// Mitsubishi GX Works2 project: 42015005-기말1   PLC: Q02/Q02H

PROGRAM MAIN
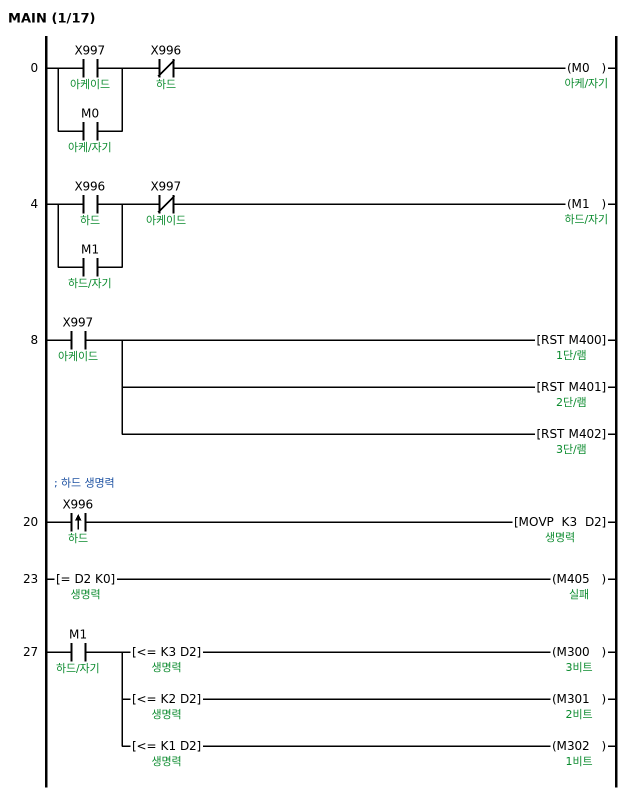
0     LD      X997  ; 아케이드
      OR      M0  ; 아케/자기
      ANI     X996  ; 하드
      OUT     M0  ; 아케/자기
4     LD      X996  ; 하드
      OR      M1  ; 하드/자기
      ANI     X997  ; 아케이드
      OUT     M1  ; 하드/자기
8     LD      X997  ; 아케이드
      RST     M400  ; 1단/램
      RST     M401  ; 2단/램
      RST     M402  ; 3단/램
; 하드 생명력
20    LDP     X996  ; 하드
      MOVP    K3 D2  ; 생명력
23    LD=     D2 K0  ; 생명력
      OUT     M405  ; 실패
27    LD      M1  ; 하드/자기
      MPS
      AND<=   K3 D2  ; 생명력
      OUT     M300  ; 3비트
      MRD
      AND<=   K2 D2  ; 생명력
      OUT     M301  ; 2비트
      MPP
      AND<=   K1 D2  ; 생명력
      OUT     M302  ; 1비트
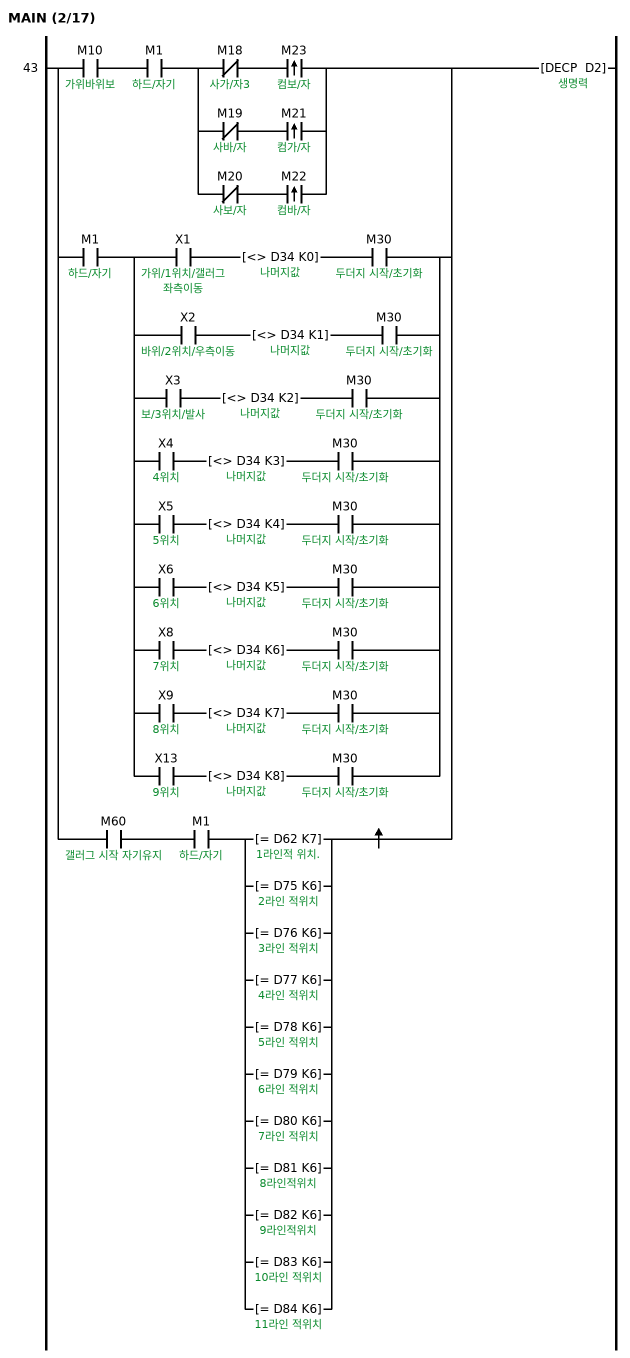
43    LD      M10  ; 가위바위보
      AND     M1  ; 하드/자기
      LDI     M18  ; 사가/자3
      ANDP    M23  ; 컴보/자
      LDI     M19  ; 사바/자
      ANDP    M21  ; 컴가/자
      ORB
      LDI     M20  ; 사보/자
      ANDP    M22  ; 컴바/자
      ORB
      ANB
      LD      M1  ; 하드/자기
      LD      X1  ; 가위/1위치/갤러그 좌측이동
      AND<>   D34 K0  ; 나머지값
      AND     M30  ; 두더지 시작/초기화
      LD      X2  ; 바위/2위치/우측이동
      AND<>   D34 K1  ; 나머지값
      AND     M30  ; 두더지 시작/초기화
      ORB
      LD      X3  ; 보/3위치/발사
      AND<>   D34 K2  ; 나머지값
      AND     M30  ; 두더지 시작/초기화
      ORB
      LD      X4  ; 4위치
      AND<>   D34 K3  ; 나머지값
      AND     M30  ; 두더지 시작/초기화
      ORB
      LD      X5  ; 5위치
      AND<>   D34 K4  ; 나머지값
      AND     M30  ; 두더지 시작/초기화
      ORB
      LD      X6  ; 6위치
      AND<>   D34 K5  ; 나머지값
      AND     M30  ; 두더지 시작/초기화
      ORB
      LD      X8  ; 7위치
      AND<>   D34 K6  ; 나머지값
      AND     M30  ; 두더지 시작/초기화
      ORB
      LD      X9  ; 8위치
      AND<>   D34 K7  ; 나머지값
      AND     M30  ; 두더지 시작/초기화
      ORB
      LD      X13  ; 9위치
      AND<>   D34 K8  ; 나머지값
      AND     M30  ; 두더지 시작/초기화
      ORB
      ANB
      ORB
      LD      M60  ; 갤러그 시작 자기유지
      AND     M1  ; 하드/자기
      LD=     D62 K7  ; 1라인적 위치.
      OR=     D75 K6  ; 2라인 적위치
      OR=     D76 K6  ; 3라인 적위치
      OR=     D77 K6  ; 4라인 적위치
      OR=     D78 K6  ; 5라인 적위치
      OR=     D79 K6  ; 6라인 적위치
      OR=     D80 K6  ; 7라인 적위치
      OR=     D81 K6  ; 8라인적위치
      OR=     D82 K6  ; 9라인적위치
      OR=     D83 K6  ; 10라인 적위치
      OR=     D84 K6  ; 11라인 적위치
      ANB
      MEP
      ORB
      DECP    D2
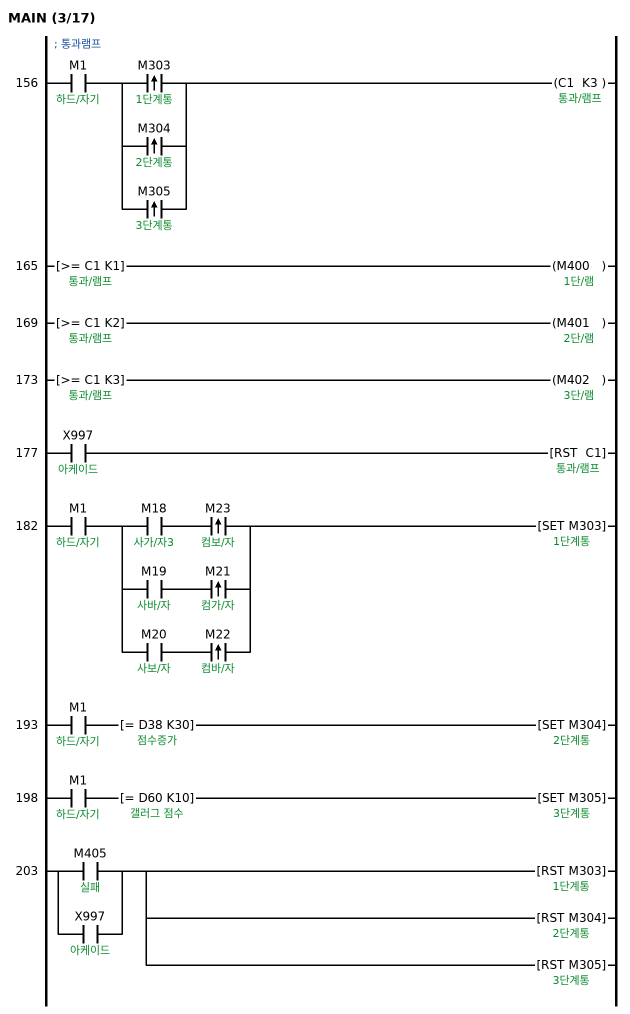
; 통과램프
156   LD      M1  ; 하드/자기
      LDP     M303  ; 1단계통
      ORP     M304  ; 2단계통
      ORP     M305  ; 3단계통
      ANB
      OUT     C1 K3  ; 통과/램프
165   LD>=    C1 K1  ; 통과/램프
      OUT     M400  ; 1단/램
169   LD>=    C1 K2  ; 통과/램프
      OUT     M401  ; 2단/램
173   LD>=    C1 K3  ; 통과/램프
      OUT     M402  ; 3단/램
177   LD      X997  ; 아케이드
      RST     C1  ; 통과/램프
182   LD      M1  ; 하드/자기
      LD      M18  ; 사가/자3
      ANDP    M23  ; 컴보/자
      LD      M19  ; 사바/자
      ANDP    M21  ; 컴가/자
      ORB
      LD      M20  ; 사보/자
      ANDP    M22  ; 컴바/자
      ORB
      ANB
      SET     M303  ; 1단계통
193   LD      M1  ; 하드/자기
      AND=    D38 K30  ; 점수증가
      SET     M304  ; 2단계통
198   LD      M1  ; 하드/자기
      AND=    D60 K10  ; 갤러그 점수
      SET     M305  ; 3단계통
203   LD      M405  ; 실패
      OR      X997  ; 아케이드
      RST     M303  ; 1단계통
      RST     M304  ; 2단계통
      RST     M305  ; 3단계통
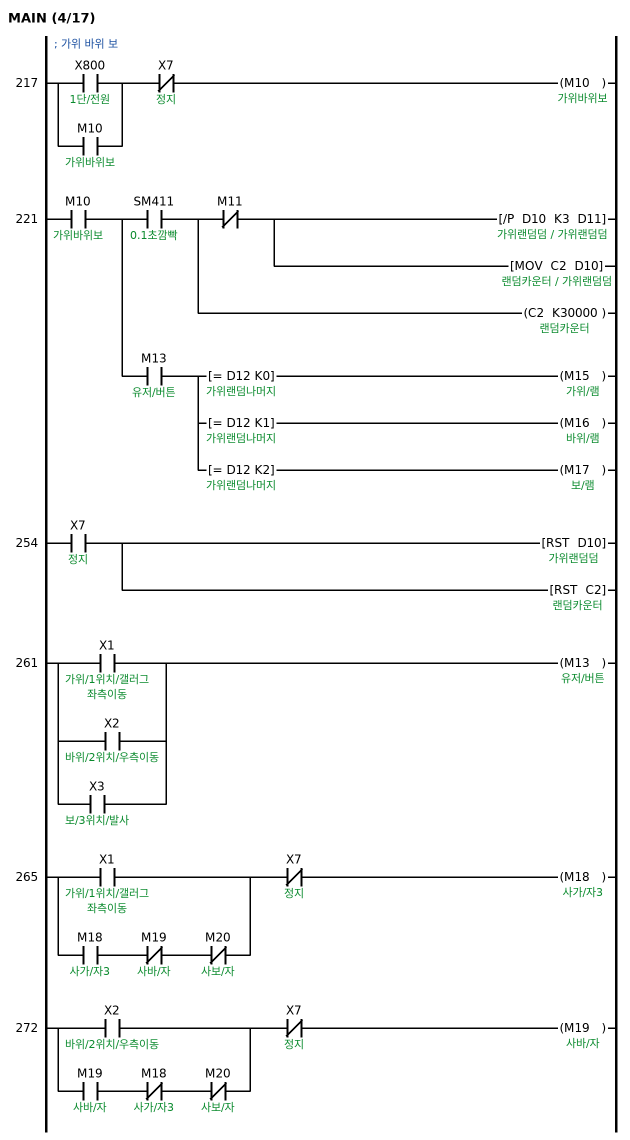
; 가위 바위 보
217   LD      X800  ; 1단/전원
      OR      M10  ; 가위바위보
      ANI     X7  ; 정지
      OUT     M10  ; 가위바위보
221   LD      M10  ; 가위바위보
      MPS
      AND     SM411  ; 0.1초깜빡
      MPS
      ANI     M11
      /P      D10 K3 D11  ; 가위랜덤덤 / 가위랜덤덤
      MOV     C2 D10  ; 랜덤카운터
      MPP
      OUT     C2 K30000  ; 랜덤카운터
      MPP
      AND     M13  ; 유저/버튼
      MPS
      AND=    D12 K0  ; 가위랜덤나머지
      OUT     M15  ; 가위/램
      MRD
      AND=    D12 K1  ; 가위랜덤나머지
      OUT     M16  ; 바위/램
      MPP
      AND=    D12 K2  ; 가위랜덤나머지
      OUT     M17  ; 보/램
254   LD      X7  ; 정지
      RST     D10  ; 가위랜덤덤
      RST     C2  ; 랜덤카운터
261   LD      X1  ; 가위/1위치/갤러그 좌측이동
      OR      X2  ; 바위/2위치/우측이동
      OR      X3  ; 보/3위치/발사
      OUT     M13  ; 유저/버튼
265   LD      X1  ; 가위/1위치/갤러그 좌측이동
      LD      M18  ; 사가/자3
      ANI     M19  ; 사바/자
      ANI     M20  ; 사보/자
      ORB
      ANI     X7  ; 정지
      OUT     M18  ; 사가/자3
272   LD      X2  ; 바위/2위치/우측이동
      LD      M19  ; 사바/자
      ANI     M18  ; 사가/자3
      ANI     M20  ; 사보/자
      ORB
      ANI     X7  ; 정지
      OUT     M19  ; 사바/자
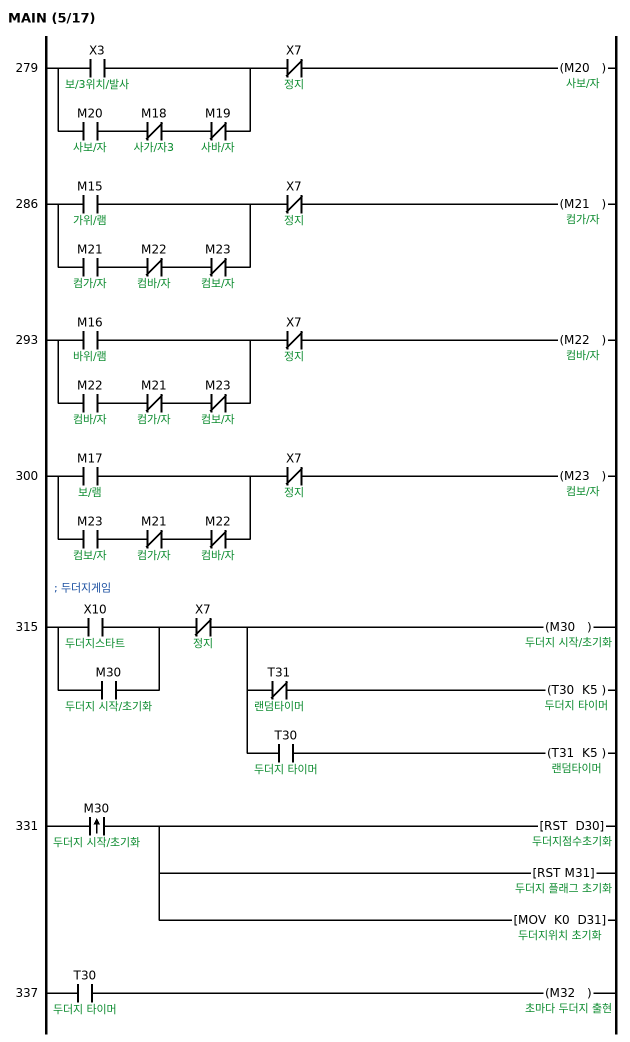
279   LD      X3  ; 보/3위치/발사
      LD      M20  ; 사보/자
      ANI     M18  ; 사가/자3
      ANI     M19  ; 사바/자
      ORB
      ANI     X7  ; 정지
      OUT     M20  ; 사보/자
286   LD      M15  ; 가위/램
      LD      M21  ; 컴가/자
      ANI     M22  ; 컴바/자
      ANI     M23  ; 컴보/자
      ORB
      ANI     X7  ; 정지
      OUT     M21  ; 컴가/자
293   LD      M16  ; 바위/램
      LD      M22  ; 컴바/자
      ANI     M21  ; 컴가/자
      ANI     M23  ; 컴보/자
      ORB
      ANI     X7  ; 정지
      OUT     M22  ; 컴바/자
300   LD      M17  ; 보/램
      LD      M23  ; 컴보/자
      ANI     M21  ; 컴가/자
      ANI     M22  ; 컴바/자
      ORB
      ANI     X7  ; 정지
      OUT     M23  ; 컴보/자
; 두더지게임
315   LD      X10  ; 두더지스타트
      OR      M30  ; 두더지 시작/초기화
      ANI     X7  ; 정지
      OUT     M30  ; 두더지 시작/초기화
      MPS
      ANI     T31  ; 랜덤타이머
      OUT     T30 K5  ; 두더지 타이머
      MPP
      AND     T30  ; 두더지 타이머
      OUT     T31 K5  ; 랜덤타이머
331   LDP     M30  ; 두더지 시작/초기화
      RST     D30  ; 두더지점수초기화
      RST     M31  ; 두더지 플래그 초기화
      MOV     K0 D31  ; 두더지위치 초기화
337   LD      T30  ; 두더지 타이머
      OUT     M32  ; 초마다 두더지 출현
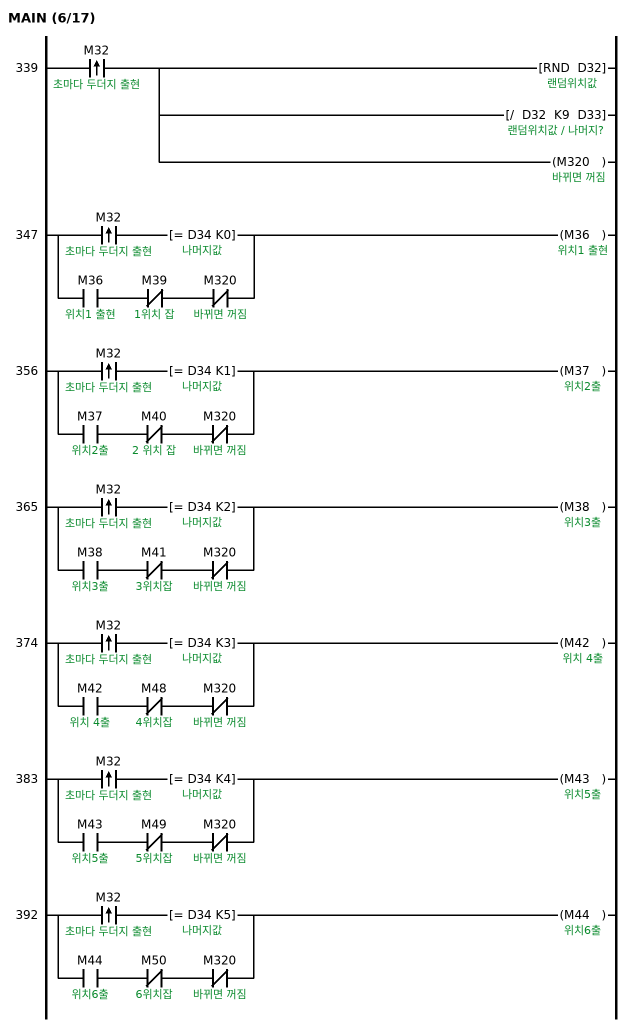
339   LDP     M32  ; 초마다 두더지 출현
      RND     D32  ; 랜덤위치값
      /       D32 K9 D33  ; 나머지?
      OUT     M320  ; 바뀌면 꺼짐
347   LDP     M32  ; 초마다 두더지 출현
      AND=    D34 K0  ; 나머지값
      LD      M36  ; 위치1 출현
      ANI     M39  ; 1위치 잡
      ANI     M320  ; 바뀌면 꺼짐
      ORB
      OUT     M36  ; 위치1 출현
356   LDP     M32  ; 초마다 두더지 출현
      AND=    D34 K1  ; 나머지값
      LD      M37  ; 위치2출
      ANI     M40  ; 2 위치 잡
      ANI     M320  ; 바뀌면 꺼짐
      ORB
      OUT     M37  ; 위치2출
365   LDP     M32  ; 초마다 두더지 출현
      AND=    D34 K2  ; 나머지값
      LD      M38  ; 위치3출
      ANI     M41  ; 3위치잡
      ANI     M320  ; 바뀌면 꺼짐
      ORB
      OUT     M38  ; 위치3출
374   LDP     M32  ; 초마다 두더지 출현
      AND=    D34 K3  ; 나머지값
      LD      M42  ; 위치 4출
      ANI     M48  ; 4위치잡
      ANI     M320  ; 바뀌면 꺼짐
      ORB
      OUT     M42  ; 위치 4출
383   LDP     M32  ; 초마다 두더지 출현
      AND=    D34 K4  ; 나머지값
      LD      M43  ; 위치5출
      ANI     M49  ; 5위치잡
      ANI     M320  ; 바뀌면 꺼짐
      ORB
      OUT     M43  ; 위치5출
392   LDP     M32  ; 초마다 두더지 출현
      AND=    D34 K5  ; 나머지값
      LD      M44  ; 위치6출
      ANI     M50  ; 6위치잡
      ANI     M320  ; 바뀌면 꺼짐
      ORB
      OUT     M44  ; 위치6출
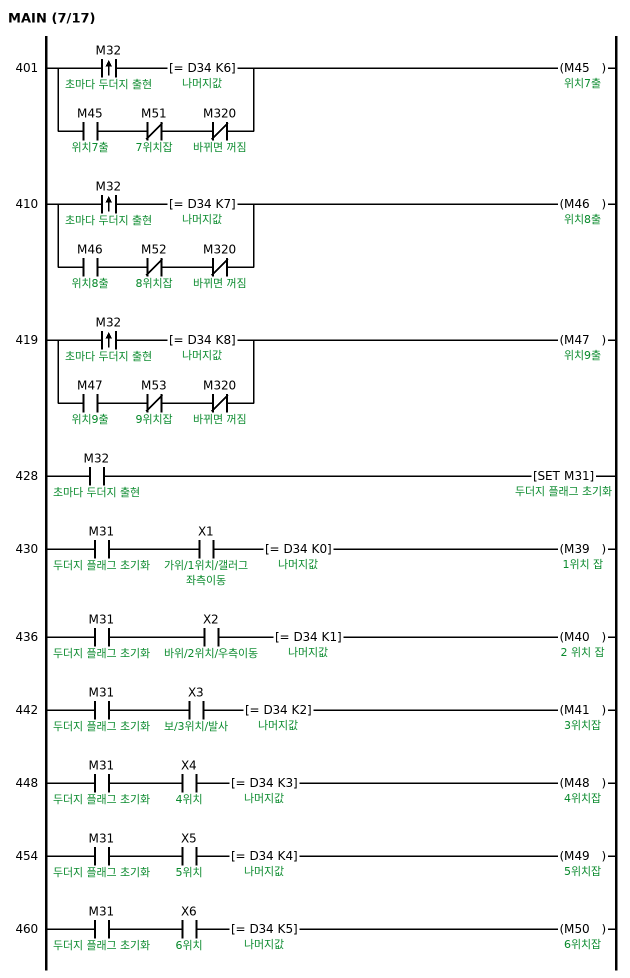
401   LDP     M32  ; 초마다 두더지 출현
      AND=    D34 K6  ; 나머지값
      LD      M45  ; 위치7출
      ANI     M51  ; 7위치잡
      ANI     M320  ; 바뀌면 꺼짐
      ORB
      OUT     M45  ; 위치7출
410   LDP     M32  ; 초마다 두더지 출현
      AND=    D34 K7  ; 나머지값
      LD      M46  ; 위치8출
      ANI     M52  ; 8위치잡
      ANI     M320  ; 바뀌면 꺼짐
      ORB
      OUT     M46  ; 위치8출
419   LDP     M32  ; 초마다 두더지 출현
      AND=    D34 K8  ; 나머지값
      LD      M47  ; 위치9출
      ANI     M53  ; 9위치잡
      ANI     M320  ; 바뀌면 꺼짐
      ORB
      OUT     M47  ; 위치9출
428   LD      M32  ; 초마다 두더지 출현
      SET     M31  ; 두더지 플래그 초기화
430   LD      M31  ; 두더지 플래그 초기화
      AND     X1  ; 가위/1위치/갤러그 좌측이동
      AND=    D34 K0  ; 나머지값
      OUT     M39  ; 1위치 잡
436   LD      M31  ; 두더지 플래그 초기화
      AND     X2  ; 바위/2위치/우측이동
      AND=    D34 K1  ; 나머지값
      OUT     M40  ; 2 위치 잡
442   LD      M31  ; 두더지 플래그 초기화
      AND     X3  ; 보/3위치/발사
      AND=    D34 K2  ; 나머지값
      OUT     M41  ; 3위치잡
448   LD      M31  ; 두더지 플래그 초기화
      AND     X4  ; 4위치
      AND=    D34 K3  ; 나머지값
      OUT     M48  ; 4위치잡
454   LD      M31  ; 두더지 플래그 초기화
      AND     X5  ; 5위치
      AND=    D34 K4  ; 나머지값
      OUT     M49  ; 5위치잡
460   LD      M31  ; 두더지 플래그 초기화
      AND     X6  ; 6위치
      AND=    D34 K5  ; 나머지값
      OUT     M50  ; 6위치잡
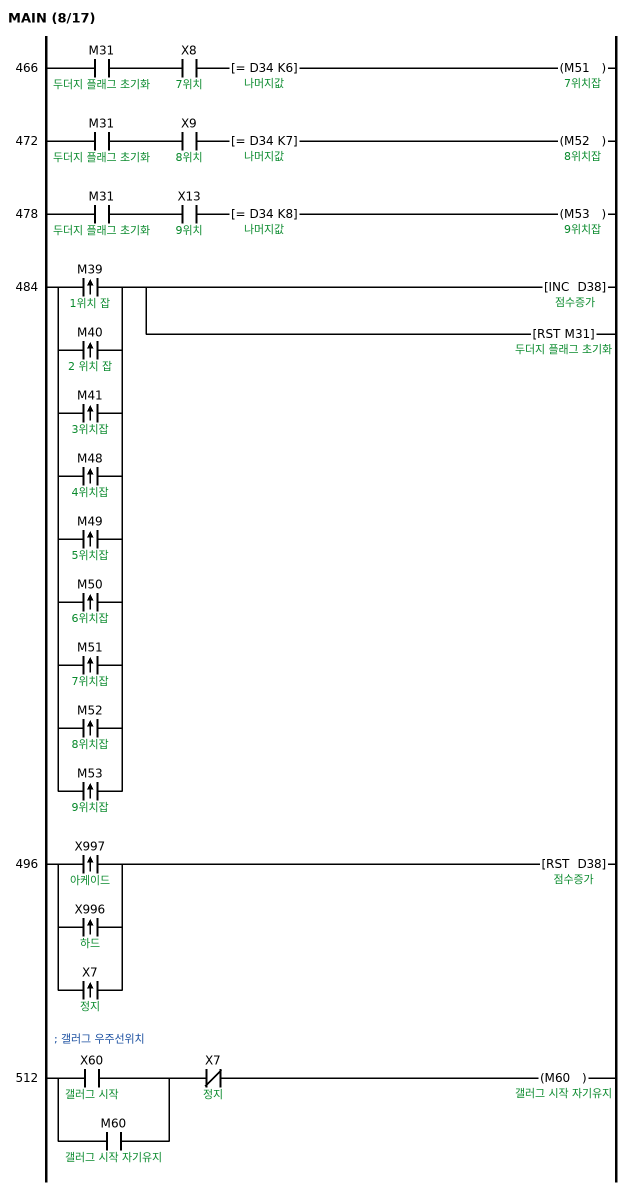
466   LD      M31  ; 두더지 플래그 초기화
      AND     X8  ; 7위치
      AND=    D34 K6  ; 나머지값
      OUT     M51  ; 7위치잡
472   LD      M31  ; 두더지 플래그 초기화
      AND     X9  ; 8위치
      AND=    D34 K7  ; 나머지값
      OUT     M52  ; 8위치잡
478   LD      M31  ; 두더지 플래그 초기화
      AND     X13  ; 9위치
      AND=    D34 K8  ; 나머지값
      OUT     M53  ; 9위치잡
484   LDP     M39  ; 1위치 잡
      ORP     M40  ; 2 위치 잡
      ORP     M41  ; 3위치잡
      ORP     M48  ; 4위치잡
      ORP     M49  ; 5위치잡
      ORP     M50  ; 6위치잡
      ORP     M51  ; 7위치잡
      ORP     M52  ; 8위치잡
      ORP     M53  ; 9위치잡
      INC     D38
      RST     M31  ; 두더지 플래그 초기화
496   LDP     X997  ; 아케이드
      ORP     X996  ; 하드
      ORP     X7  ; 정지
      RST     D38  ; 점수증가
; 갤러그 우주선위치
512   LD      X60  ; 갤러그 시작
      OR      M60  ; 갤러그 시작 자기유지
      ANI     X7  ; 정지
      OUT     M60  ; 갤러그 시작 자기유지
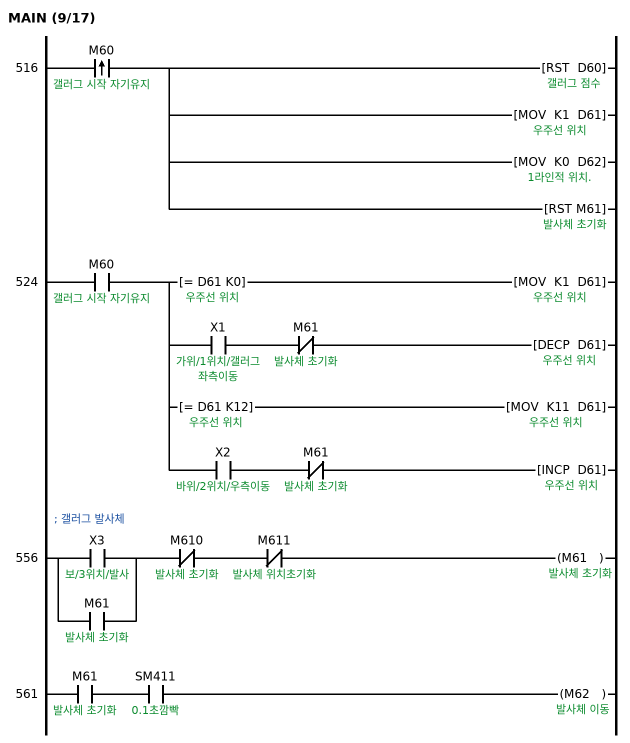
516   LDP     M60  ; 갤러그 시작 자기유지
      RST     D60  ; 갤러그 점수
      MOV     K1 D61  ; 우주선 위치
      MOV     K0 D62
      RST     M61  ; 발사체 초기화
524   LD      M60  ; 갤러그 시작 자기유지
      MPS
      AND=    D61 K0  ; 우주선 위치
      MOV     K1 D61
      MRD
      AND     X1  ; 가위/1위치/갤러그 좌측이동
      ANI     M61  ; 발사체 초기화
      DECP    D61
      MRD
      AND=    D61 K12  ; 우주선 위치
      MOV     K11 D61
      MPP
      AND     X2  ; 바위/2위치/우측이동
      ANI     M61  ; 발사체 초기화
      INCP    D61
; 갤러그 발사체
556   LD      X3  ; 보/3위치/발사
      OR      M61  ; 발사체 초기화
      ANI     M610  ; 발사체 초기화
      ANI     M611  ; 발사체 위치초기화
      OUT     M61  ; 발사체 초기화
561   LD      M61  ; 발사체 초기화
      AND     SM411  ; 0.1초깜빡
      OUT     M62  ; 발사체 이동
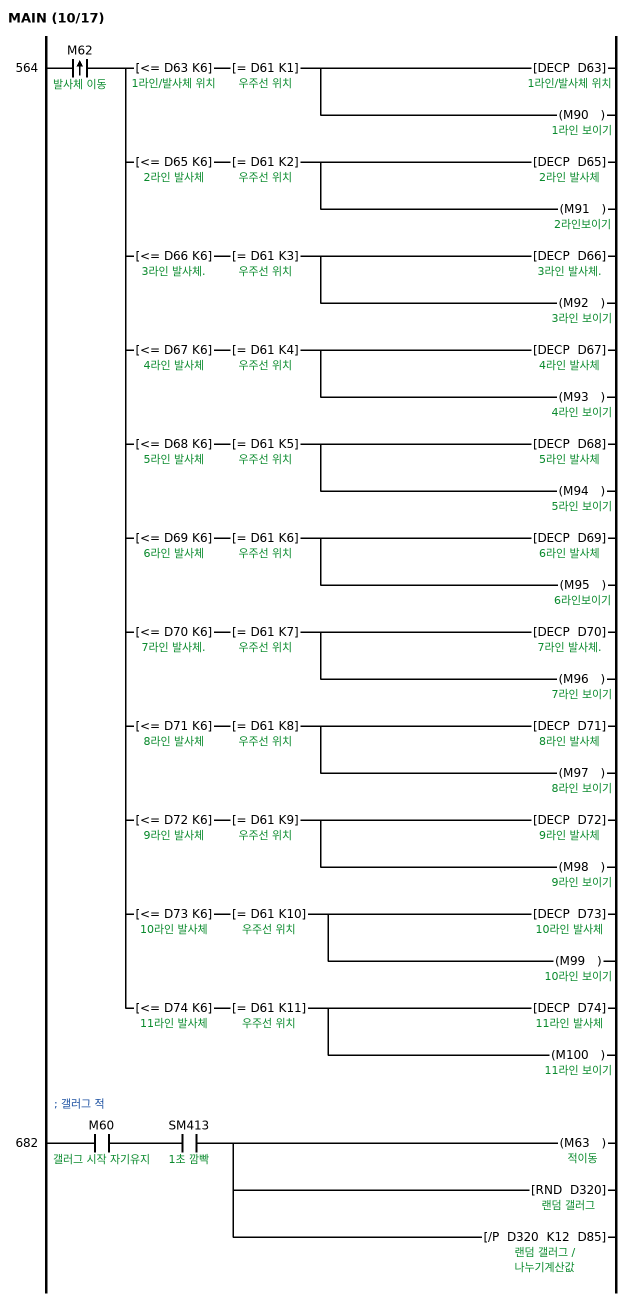
564   LDP     M62  ; 발사체 이동
      MPS
      AND<=   D63 K6  ; 1라인/발사체 위치
      AND=    D61 K1  ; 우주선 위치
      DECP    D63
      OUT     M90  ; 1라인 보이기
      MRD
      AND<=   D65 K6  ; 2라인 발사체
      AND=    D61 K2  ; 우주선 위치
      DECP    D65
      OUT     M91  ; 2라인보이기
      MRD
      AND<=   D66 K6  ; 3라인 발사체.
      AND=    D61 K3  ; 우주선 위치
      DECP    D66
      OUT     M92  ; 3라인 보이기
      MRD
      AND<=   D67 K6  ; 4라인 발사체
      AND=    D61 K4  ; 우주선 위치
      DECP    D67
      OUT     M93  ; 4라인 보이기
      MRD
      AND<=   D68 K6  ; 5라인 발사체
      AND=    D61 K5  ; 우주선 위치
      DECP    D68
      OUT     M94  ; 5라인 보이기
      MRD
      AND<=   D69 K6  ; 6라인 발사체
      AND=    D61 K6  ; 우주선 위치
      DECP    D69
      OUT     M95  ; 6라인보이기
      MRD
      AND<=   D70 K6  ; 7라인 발사체.
      AND=    D61 K7  ; 우주선 위치
      DECP    D70
      OUT     M96  ; 7라인 보이기
      MRD
      AND<=   D71 K6  ; 8라인 발사체
      AND=    D61 K8  ; 우주선 위치
      DECP    D71
      OUT     M97  ; 8라인 보이기
      MRD
      AND<=   D72 K6  ; 9라인 발사체
      AND=    D61 K9  ; 우주선 위치
      DECP    D72
      OUT     M98  ; 9라인 보이기
      MRD
      AND<=   D73 K6  ; 10라인 발사체
      AND=    D61 K10  ; 우주선 위치
      DECP    D73
      OUT     M99  ; 10라인 보이기
      MPP
      AND<=   D74 K6  ; 11라인 발사체
      AND=    D61 K11  ; 우주선 위치
      DECP    D74
      OUT     M100  ; 11라인 보이기
; 갤러그 적
682   LD      M60  ; 갤러그 시작 자기유지
      AND     SM413  ; 1초 깜빡
      OUT     M63  ; 적이동
      RND     D320  ; 랜덤 갤러그
      /P      D320 K12 D85  ; 나누기계산값
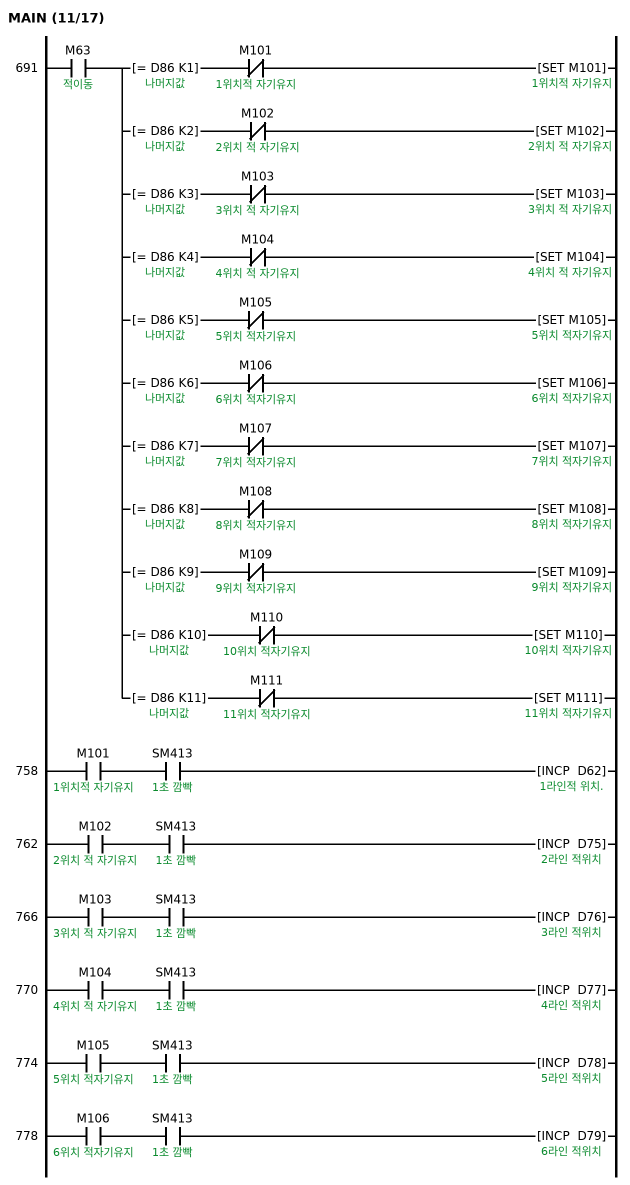
691   LD      M63  ; 적이동
      MPS
      AND=    D86 K1  ; 나머지값
      ANI     M101  ; 1위치적 자기유지
      SET     M101  ; 1위치적 자기유지
      MRD
      AND=    D86 K2  ; 나머지값
      ANI     M102  ; 2위치 적 자기유지
      SET     M102  ; 2위치 적 자기유지
      MRD
      AND=    D86 K3  ; 나머지값
      ANI     M103  ; 3위치 적 자기유지
      SET     M103  ; 3위치 적 자기유지
      MRD
      AND=    D86 K4  ; 나머지값
      ANI     M104  ; 4위치 적 자기유지
      SET     M104  ; 4위치 적 자기유지
      MRD
      AND=    D86 K5  ; 나머지값
      ANI     M105  ; 5위치 적자기유지
      SET     M105  ; 5위치 적자기유지
      MRD
      AND=    D86 K6  ; 나머지값
      ANI     M106  ; 6위치 적자기유지
      SET     M106  ; 6위치 적자기유지
      MRD
      AND=    D86 K7  ; 나머지값
      ANI     M107  ; 7위치 적자기유지
      SET     M107  ; 7위치 적자기유지
      MRD
      AND=    D86 K8  ; 나머지값
      ANI     M108  ; 8위치 적자기유지
      SET     M108  ; 8위치 적자기유지
      MRD
      AND=    D86 K9  ; 나머지값
      ANI     M109  ; 9위치 적자기유지
      SET     M109  ; 9위치 적자기유지
      MRD
      AND=    D86 K10  ; 나머지값
      ANI     M110  ; 10위치 적자기유지
      SET     M110  ; 10위치 적자기유지
      MPP
      AND=    D86 K11  ; 나머지값
      ANI     M111  ; 11위치 적자기유지
      SET     M111  ; 11위치 적자기유지
758   LD      M101  ; 1위치적 자기유지
      AND     SM413  ; 1초 깜빡
      INCP    D62
762   LD      M102  ; 2위치 적 자기유지
      AND     SM413  ; 1초 깜빡
      INCP    D75
766   LD      M103  ; 3위치 적 자기유지
      AND     SM413  ; 1초 깜빡
      INCP    D76
770   LD      M104  ; 4위치 적 자기유지
      AND     SM413  ; 1초 깜빡
      INCP    D77
774   LD      M105  ; 5위치 적자기유지
      AND     SM413  ; 1초 깜빡
      INCP    D78
778   LD      M106  ; 6위치 적자기유지
      AND     SM413  ; 1초 깜빡
      INCP    D79
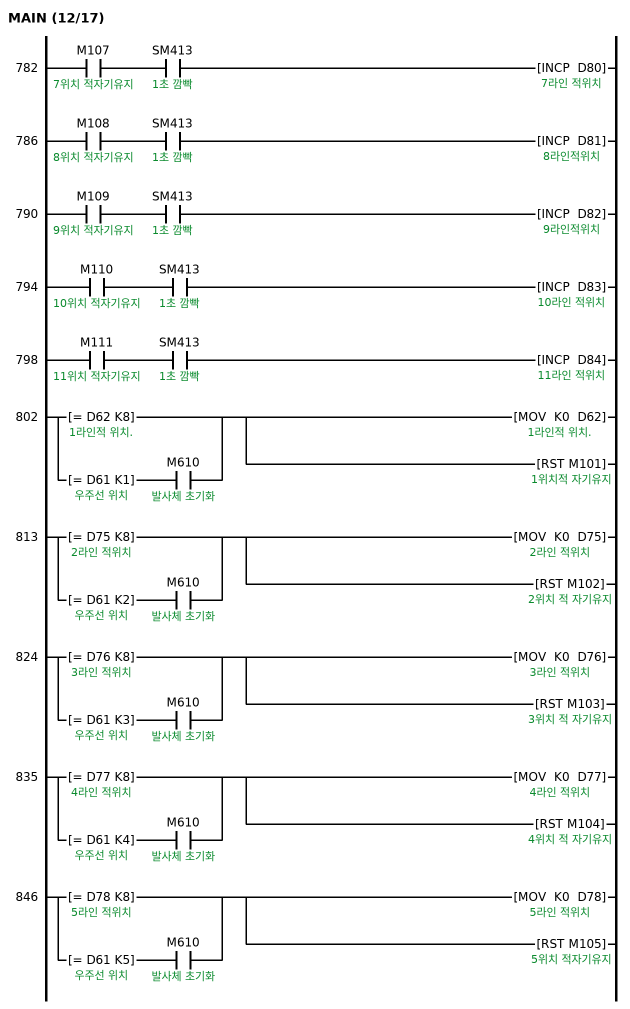
782   LD      M107  ; 7위치 적자기유지
      AND     SM413  ; 1초 깜빡
      INCP    D80
786   LD      M108  ; 8위치 적자기유지
      AND     SM413  ; 1초 깜빡
      INCP    D81
790   LD      M109  ; 9위치 적자기유지
      AND     SM413  ; 1초 깜빡
      INCP    D82
794   LD      M110  ; 10위치 적자기유지
      AND     SM413  ; 1초 깜빡
      INCP    D83
798   LD      M111  ; 11위치 적자기유지
      AND     SM413  ; 1초 깜빡
      INCP    D84
802   LD=     D62 K8  ; 1라인적 위치.
      LD=     D61 K1  ; 우주선 위치
      AND     M610  ; 발사체 초기화
      ORB
      MOV     K0 D62
      RST     M101  ; 1위치적 자기유지
813   LD=     D75 K8  ; 2라인 적위치
      LD=     D61 K2  ; 우주선 위치
      AND     M610  ; 발사체 초기화
      ORB
      MOV     K0 D75
      RST     M102  ; 2위치 적 자기유지
824   LD=     D76 K8  ; 3라인 적위치
      LD=     D61 K3  ; 우주선 위치
      AND     M610  ; 발사체 초기화
      ORB
      MOV     K0 D76
      RST     M103  ; 3위치 적 자기유지
835   LD=     D77 K8  ; 4라인 적위치
      LD=     D61 K4  ; 우주선 위치
      AND     M610  ; 발사체 초기화
      ORB
      MOV     K0 D77
      RST     M104  ; 4위치 적 자기유지
846   LD=     D78 K8  ; 5라인 적위치
      LD=     D61 K5  ; 우주선 위치
      AND     M610  ; 발사체 초기화
      ORB
      MOV     K0 D78
      RST     M105  ; 5위치 적자기유지
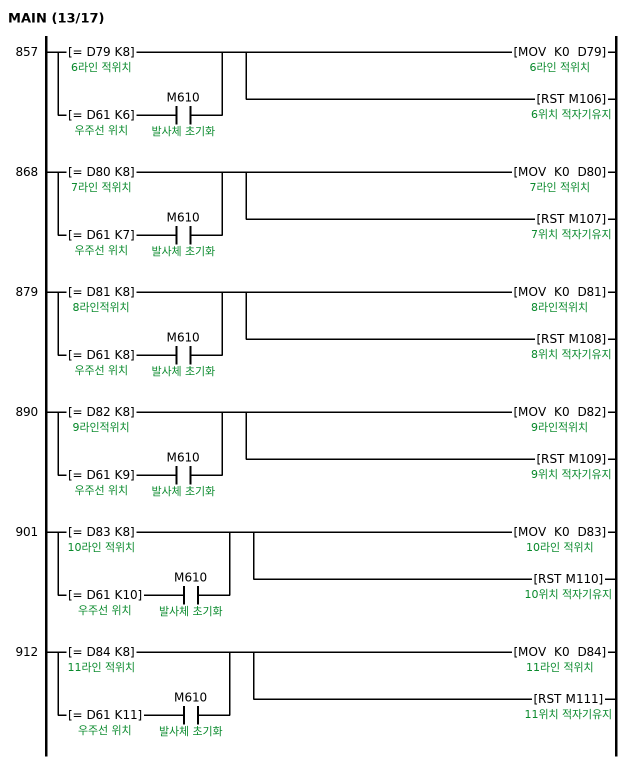
857   LD=     D79 K8  ; 6라인 적위치
      LD=     D61 K6  ; 우주선 위치
      AND     M610  ; 발사체 초기화
      ORB
      MOV     K0 D79
      RST     M106  ; 6위치 적자기유지
868   LD=     D80 K8  ; 7라인 적위치
      LD=     D61 K7  ; 우주선 위치
      AND     M610  ; 발사체 초기화
      ORB
      MOV     K0 D80
      RST     M107  ; 7위치 적자기유지
879   LD=     D81 K8  ; 8라인적위치
      LD=     D61 K8  ; 우주선 위치
      AND     M610  ; 발사체 초기화
      ORB
      MOV     K0 D81
      RST     M108  ; 8위치 적자기유지
890   LD=     D82 K8  ; 9라인적위치
      LD=     D61 K9  ; 우주선 위치
      AND     M610  ; 발사체 초기화
      ORB
      MOV     K0 D82
      RST     M109  ; 9위치 적자기유지
901   LD=     D83 K8  ; 10라인 적위치
      LD=     D61 K10  ; 우주선 위치
      AND     M610  ; 발사체 초기화
      ORB
      MOV     K0 D83
      RST     M110  ; 10위치 적자기유지
912   LD=     D84 K8  ; 11라인 적위치
      LD=     D61 K11  ; 우주선 위치
      AND     M610  ; 발사체 초기화
      ORB
      MOV     K0 D84
      RST     M111  ; 11위치 적자기유지
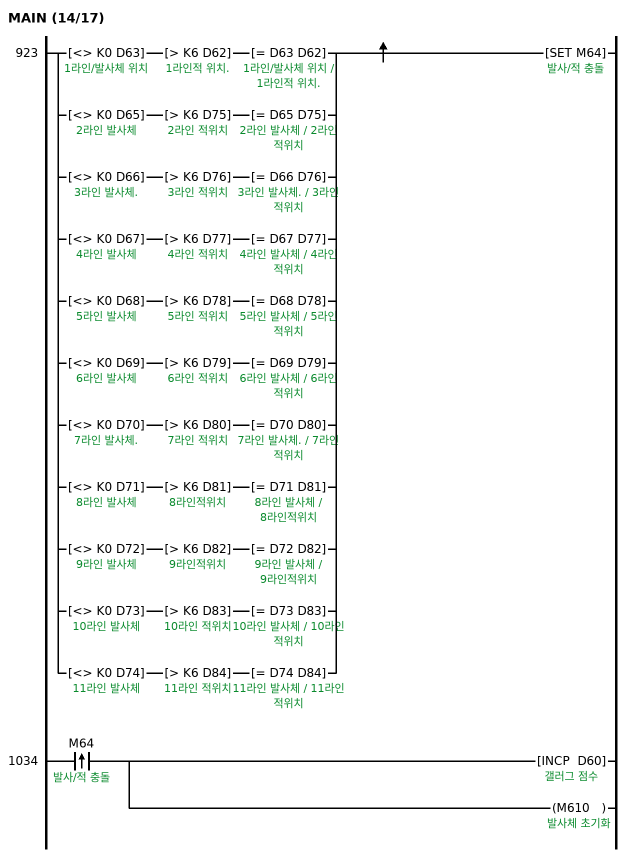
923   LD<>    K0 D63  ; 1라인/발사체 위치
      AND>    K6 D62  ; 1라인적 위치.
      AND=    D63 D62  ; 1라인/발사체 위치 / 1라인적 위치.
      LD<>    K0 D65  ; 2라인 발사체
      AND>    K6 D75  ; 2라인 적위치
      AND=    D65 D75  ; 2라인 발사체 / 2라인 적위치
      ORB
      LD<>    K0 D66  ; 3라인 발사체.
      AND>    K6 D76  ; 3라인 적위치
      AND=    D66 D76  ; 3라인 발사체. / 3라인 적위치
      ORB
      LD<>    K0 D67  ; 4라인 발사체
      AND>    K6 D77  ; 4라인 적위치
      AND=    D67 D77  ; 4라인 발사체 / 4라인 적위치
      ORB
      LD<>    K0 D68  ; 5라인 발사체
      AND>    K6 D78  ; 5라인 적위치
      AND=    D68 D78  ; 5라인 발사체 / 5라인 적위치
      ORB
      LD<>    K0 D69  ; 6라인 발사체
      AND>    K6 D79  ; 6라인 적위치
      AND=    D69 D79  ; 6라인 발사체 / 6라인 적위치
      ORB
      LD<>    K0 D70  ; 7라인 발사체.
      AND>    K6 D80  ; 7라인 적위치
      AND=    D70 D80  ; 7라인 발사체. / 7라인 적위치
      ORB
      LD<>    K0 D71  ; 8라인 발사체
      AND>    K6 D81  ; 8라인적위치
      AND=    D71 D81  ; 8라인 발사체 / 8라인적위치
      ORB
      LD<>    K0 D72  ; 9라인 발사체
      AND>    K6 D82  ; 9라인적위치
      AND=    D72 D82  ; 9라인 발사체 / 9라인적위치
      ORB
      LD<>    K0 D73  ; 10라인 발사체
      AND>    K6 D83  ; 10라인 적위치
      AND=    D73 D83  ; 10라인 발사체 / 10라인 적위치
      ORB
      LD<>    K0 D74  ; 11라인 발사체
      AND>    K6 D84  ; 11라인 적위치
      AND=    D74 D84  ; 11라인 발사체 / 11라인 적위치
      ORB
      MEP
      SET     M64  ; 발사/적 충돌
1034  LDP     M64  ; 발사/적 충돌
      INCP    D60
      OUT     M610  ; 발사체 초기화
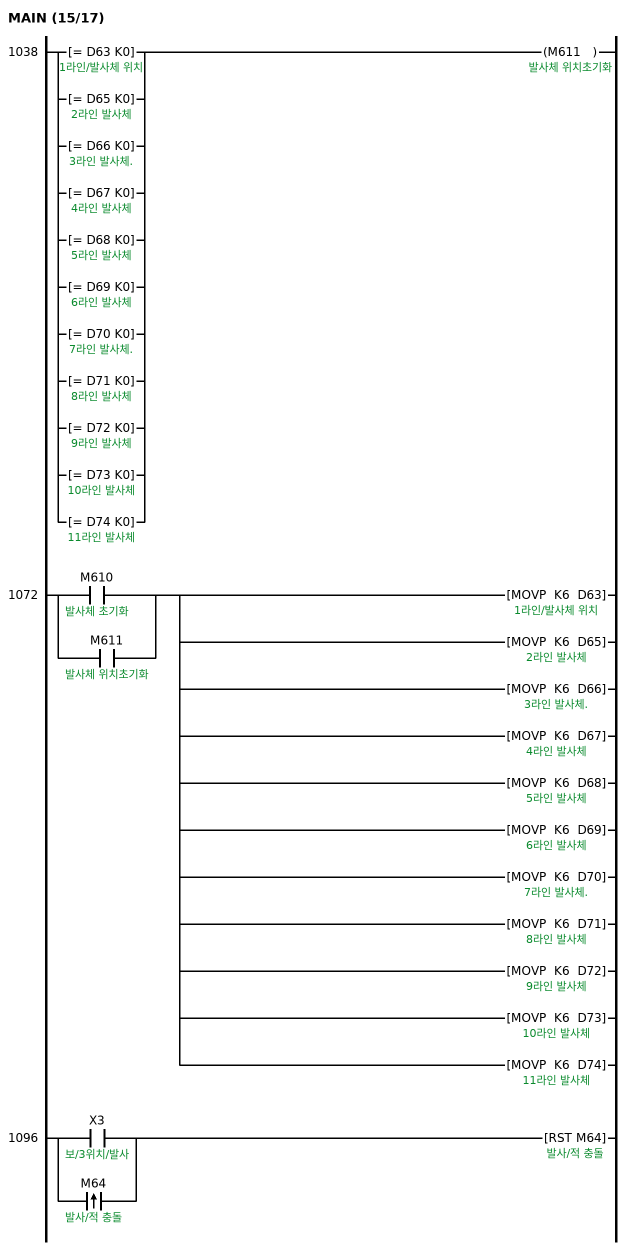
1038  LD=     D63 K0  ; 1라인/발사체 위치
      OR=     D65 K0  ; 2라인 발사체
      OR=     D66 K0  ; 3라인 발사체.
      OR=     D67 K0  ; 4라인 발사체
      OR=     D68 K0  ; 5라인 발사체
      OR=     D69 K0  ; 6라인 발사체
      OR=     D70 K0  ; 7라인 발사체.
      OR=     D71 K0  ; 8라인 발사체
      OR=     D72 K0  ; 9라인 발사체
      OR=     D73 K0  ; 10라인 발사체
      OR=     D74 K0  ; 11라인 발사체
      OUT     M611  ; 발사체 위치초기화
1072  LD      M610  ; 발사체 초기화
      OR      M611  ; 발사체 위치초기화
      MOVP    K6 D63
      MOVP    K6 D65
      MOVP    K6 D66
      MOVP    K6 D67
      MOVP    K6 D68
      MOVP    K6 D69
      MOVP    K6 D70
      MOVP    K6 D71
      MOVP    K6 D72
      MOVP    K6 D73
      MOVP    K6 D74
1096  LD      X3  ; 보/3위치/발사
      ORP     M64  ; 발사/적 충돌
      RST     M64  ; 발사/적 충돌
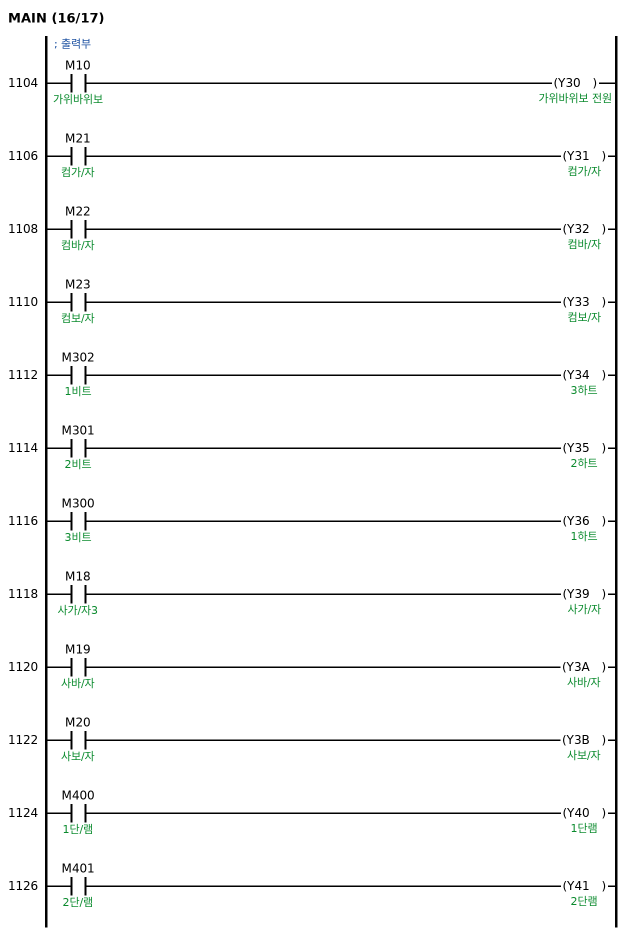
; 출력부
1104  LD      M10  ; 가위바위보
      OUT     Y30  ; 가위바위보 전원
1106  LD      M21  ; 컴가/자
      OUT     Y31  ; 컴가/자
1108  LD      M22  ; 컴바/자
      OUT     Y32  ; 컴바/자
1110  LD      M23  ; 컴보/자
      OUT     Y33  ; 컴보/자
1112  LD      M302  ; 1비트
      OUT     Y34  ; 3하트
1114  LD      M301  ; 2비트
      OUT     Y35  ; 2하트
1116  LD      M300  ; 3비트
      OUT     Y36  ; 1하트
1118  LD      M18  ; 사가/자3
      OUT     Y39  ; 사가/자
1120  LD      M19  ; 사바/자
      OUT     Y3A  ; 사바/자
1122  LD      M20  ; 사보/자
      OUT     Y3B  ; 사보/자
1124  LD      M400  ; 1단/램
      OUT     Y40  ; 1단램
1126  LD      M401  ; 2단/램
      OUT     Y41  ; 2단램
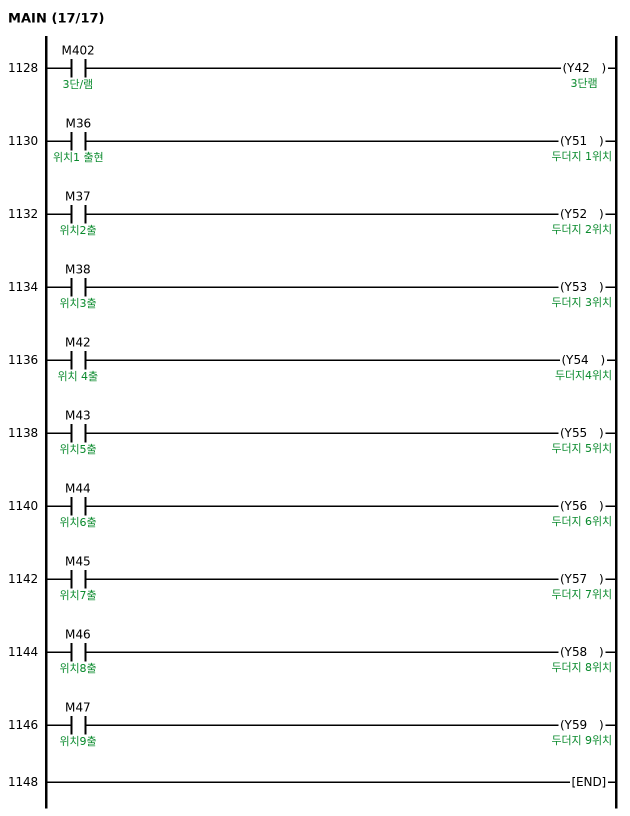
1128  LD      M402  ; 3단/램
      OUT     Y42  ; 3단램
1130  LD      M36  ; 위치1 출현
      OUT     Y51  ; 두더지 1위치
1132  LD      M37  ; 위치2출
      OUT     Y52  ; 두더지 2위치
1134  LD      M38  ; 위치3출
      OUT     Y53  ; 두더지 3위치
1136  LD      M42  ; 위치 4출
      OUT     Y54  ; 두더지4위치
1138  LD      M43  ; 위치5출
      OUT     Y55  ; 두더지 5위치
1140  LD      M44  ; 위치6출
      OUT     Y56  ; 두더지 6위치
1142  LD      M45  ; 위치7출
      OUT     Y57  ; 두더지 7위치
1144  LD      M46  ; 위치8출
      OUT     Y58  ; 두더지 8위치
1146  LD      M47  ; 위치9출
      OUT     Y59  ; 두더지 9위치
1148  END
END_PROGRAM

// device comments not shown above
X998  ; 배속
X999  ; 정속
M35  ; 랜덤 생성
M306  ; 4단계통
M307  ; 5단계통
M403  ; 4단/램
M404  ; 5단/램
D0  ; 정속값
D1  ; 배속값
D15  ; 사가
D16  ; 사바
D17  ; 사보
D18  ; 컴가
D35  ; 3 나머지값
